// TIA Portal V16 export
// export: Created 2021-09-22T13:16:19.9691537Z, ExportSetting WithDefaults, DisplayName Totally Integrated Automation Portal, DisplayVersion V16 Update 1, DisplayName TIA Portal Version Control Interface, DisplayVersion V16, DisplayName TIA Portal Openness, DisplayVersion V16, DisplayName SINAMICS Startdrive Advanced, DisplayVersion V16 Update 5, DisplayName SINAMICS Startdrive G130, G150, S120, S150, SINAMICS MV, S210, DisplayVersion V16 Update 5, DisplayName SINAMICS Startdrive G110M, G120, G120C, G120D, G120P, G115D, DisplayVersion V16 Update 5, DisplayName STEP 7 Professional, DisplayVersion V16, DisplayName STEP 7 Safety, DisplayVersion V16, DisplayName WinCC Professional, DisplayVersion V16
FUNCTION_BLOCK "FB549.Divert.Sorter.Basing"   // FB543, LAD
{ S7_Optimized_Access := 'TRUE' }
VERSION : 0.1
// stored: AutoNumber false, IsIECCheckEnabled false, IsRetainMemResEnabled false, MemoryReserve 100, SetENOAutomatically false, UDAEnableTagReadback false
   VAR_INPUT
      Acil_Yok : Bool;
      Sorter_Calisiyor : Bool;
      Sağ_Chute_Sorted_Sensoru : Bool;
      Sol_Chute_Sorted_Sensoru : Bool;
      "Sağ_Chute_Aktif / Pasif" : Bool;   // 1 = Aktif , 0 = Pasif
      "Sol_Chute_Aktif / Pasif" : Bool;   // 1 = Aktif , 0 = Pasif
      Chute_Rulo_Hatası : Bool;
      Divert_Sürücü_Hatası : Bool;
      Pozisyon_Olcme_Aktif : Bool;
      Sağ_Çıkış_Target { ExternalAccessible := 'False'; ExternalVisible := 'False'; ExternalWritable := 'False'} : Int;
      Sol_Çıkış_Target { ExternalAccessible := 'False'; ExternalVisible := 'False'; ExternalWritable := 'False'} : Int;
      CN_NO : Int;
      "Aktüel Encoder Değeri" : LReal;
      Birinci_Divert_Min : LReal;
      Birinci_Divert_Max : LReal;
      İkinci_Divert_Min : LReal;
      İkinci_Divert_Max : LReal;
      Max_Kutu_Adedi { ExternalAccessible := 'False'; ExternalVisible := 'False'; ExternalWritable := 'False'} : Int;
   END_VAR
   VAR_OUTPUT
      "1_sol_Divert_Çalıştır" : Bool;
      "2_sol_Divert_Çalıştır" : Bool;
      "1_sağ_Divert_Çalıştır" : Bool;
      "2_sağ_Divert_Çalıştır" : Bool;
      "Sort Hatası" : Bool;
   END_VAR
   VAR
      Sort_Aktif_AUX : Array[1..10] of Bool;
      Sort_Aktif_PTrig : Array[1..10] of Bool;
      TOF_TIME : Array[1..10] of TOF_TIME;
      TON_TIME { S7_SetPoint := 'True'} : Array[1..10] of TON_TIME;
      Sort_Aktif1 : Bool;
      Sort_Aktif2 : Bool;
      Sort_Aktif1_Sağ : Bool;
      Sort_Aktif2_Sağ : Bool;
      Sağ_Sort_Pasif : Bool;
      Sol_Sort_Pasif : Bool;
      Ikinci_Servo_Baslama : Time;
      Divert_Durdur : Bool;
      Sort_Aktif_1 { ExternalAccessible := 'False'; ExternalVisible := 'False'; ExternalWritable := 'False'} : Array[1..10] of Bool;
      Sort_Aktif_2 { ExternalAccessible := 'False'; ExternalVisible := 'False'; ExternalWritable := 'False'} : Array[1..10] of Bool;
      Sort_Aktif_1_Sağ : Array[1..10] of Bool;
      Sort_Aktif_2_Sağ : Array[1..10] of Bool;
      Sort_Ilk_Pozisyon { ExternalAccessible := 'False'; ExternalVisible := 'False'; ExternalWritable := 'False'} : Array[1..10] of LReal;
      Sort_Ön_Pozisyon { ExternalAccessible := 'False'; ExternalVisible := 'False'; ExternalWritable := 'False'} : Array[1..10] of LReal;
      Sort_Aktif_Boy { ExternalAccessible := 'False'; ExternalVisible := 'False'; ExternalWritable := 'False'} : Array[1..10] of LReal;
      SortKutuNo : Int;
      Target100 : Bool;
      Target200 : Bool;
   END_VAR
   VAR_TEMP
      "On/Off" : Bool;
      j : Int;
      Ekstra_Uzunluk : LReal;
   END_VAR
   VAR_TEMP   // added for the SCL form of the ladder/FBD networks
      _w1 : Bool;
      _w2 : Bool;
      _w3 : Bool;
      _w4 : Bool;
   END_VAR
BEGIN

REGION Network 1: On / Off
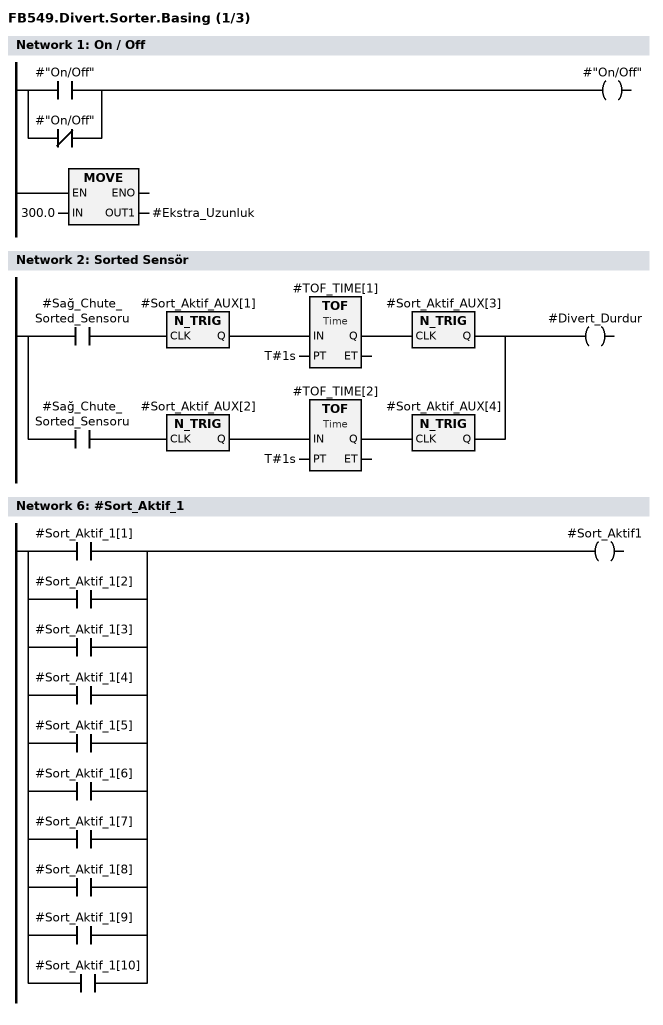
   RUNG wire#powerrail
      Contact( #"On/Off" )
      wire#w1
      Coil( #"On/Off" )
   END_RUNG
   RUNG wire#powerrail
      I_Contact( #"On/Off" )
   END_RUNG wire#w1
   RUNG wire#powerrail
      Move(in := 300.0, out1 => #Ekstra_Uzunluk)
   END_RUNG
   // the same network as SCL:
   #"On/Off" := #"On/Off" OR NOT #"On/Off";
   #Ekstra_Uzunluk := 300.0;
END_REGION

REGION Network 2: Sorted Sensör
   RUNG wire#powerrail
      Contact( #Sağ_Chute_Sorted_Sensoru )
      N_Trig( #Sort_Aktif_AUX[1] )
      { S7_Templates := "time_type := Time" } #TOF_TIME[1].TOF(pt := T#1s, et =>)
      N_Trig( #Sort_Aktif_AUX[3] )
      wire#w1
      Coil( #Divert_Durdur )
   END_RUNG
   RUNG wire#powerrail
      Contact( #Sağ_Chute_Sorted_Sensoru )
      N_Trig( #Sort_Aktif_AUX[2] )
      { S7_Templates := "time_type := Time" } #TOF_TIME[2].TOF(pt := T#1s, et =>)
      N_Trig( #Sort_Aktif_AUX[4] )
   END_RUNG wire#w1
   // the same network as SCL:
   #_w1 := NOT #Sağ_Chute_Sorted_Sensoru AND #Sort_Aktif_AUX[1];   // falling edge
   #Sort_Aktif_AUX[1] := #Sağ_Chute_Sorted_Sensoru;
   #TOF_TIME[1].TOF(IN := #_w1, PT := T#1s);
   #_w2 := NOT #TOF_TIME[1].Q AND #Sort_Aktif_AUX[3];   // falling edge
   #Sort_Aktif_AUX[3] := #TOF_TIME[1].Q;
   #_w3 := NOT #Sağ_Chute_Sorted_Sensoru AND #Sort_Aktif_AUX[2];   // falling edge
   #Sort_Aktif_AUX[2] := #Sağ_Chute_Sorted_Sensoru;
   #TOF_TIME[2].TOF(IN := #_w3, PT := T#1s);
   #_w4 := NOT #TOF_TIME[2].Q AND #Sort_Aktif_AUX[4];   // falling edge
   #Sort_Aktif_AUX[4] := #TOF_TIME[2].Q;
   #Divert_Durdur := #_w2 OR #_w4;
END_REGION

REGION Network 3 (SCL): Kutu Ön Arka Pozisyon Hesap
   // IF #Sensör.Sensor_N_Trig THEN
   //     #Sort_Ilk_Pozisyon["DB530_Kutu".CN_NO_Anlık_Kutu_Sayısı[#CN_NO]] := #"Aktüel Encoder Değeri";
   // END_IF;
   // FOR #j := 1 TO #Max_Kutu_Adedi BY 1 DO
   //     IF "DB530_Kutu".CN_NO[#CN_NO].Kutu_No[#j].VARMI = TRUE THEN
   //         #Sort_Ön_Pozisyon[#j] := #"Aktüel Encoder Değeri" - #Sort_Ilk_Pozisyon[#j];
   //     END_IF;
   // END_FOR;
END_REGION

REGION Network 4 (SCL): Sol Sort Aktif Kararı
   IF #Pozisyon_Olcme_Aktif = 0
       // AND #Sorter_Calisiyor = TRUE
       // AND #"Sol_Chute_Aktif / Pasif"
   THEN
       FOR #j := 1 TO #Max_Kutu_Adedi BY 1 DO
           IF "DB530_Kutu".CN_NO[#CN_NO].Kutu_No[#j].VARMI THEN

               IF "DB530_Kutu".CN_NO[#CN_NO].Kutu_No[#j].Target = 201
                   OR "DB530_Kutu".CN_NO[#CN_NO].Kutu_No[#j].Target = 202
                   OR "DB530_Kutu".CN_NO[#CN_NO].Kutu_No[#j].Target = 203
                   OR "DB530_Kutu".CN_NO[#CN_NO].Kutu_No[#j].Target = 204 THEN
                   #Target200 := 1;
               ELSE
                   #Target200 := 0;
               END_IF;

               IF #"Sol_Chute_Aktif / Pasif" = 1
                   AND #Chute_Rulo_Hatası = 0
                   AND #Divert_Sürücü_Hatası = 0
                   // AND #Sol_Sort_Pasif = 0
                   AND #Acil_Yok = 1
                   AND "DB530_Kutu".CN_NO[#CN_NO].Kutu_No[#j].Posizyon >= #Birinci_Divert_Min
                   AND "DB530_Kutu".CN_NO[#CN_NO].Kutu_No[#j].Posizyon <= #Birinci_Divert_Min + "DB530_Kutu".CN_NO[#CN_NO].Kutu_No[#j].Uzunluk + #Ekstra_Uzunluk
                   AND  #Target200 = 1
                   // AND "DB530_Kutu".CN_NO[#CN_NO].Kutu_No[#j].Sort_Aktifleştirildi = FALSE
               THEN
                   #Sort_Aktif_1[#j] := TRUE;
               ELSE
                   #Sort_Aktif_1[#j] := FALSE;
               END_IF;

               IF #"Sol_Chute_Aktif / Pasif" = 1
                   AND #Chute_Rulo_Hatası = 0
                   AND #Divert_Sürücü_Hatası = 0
                   // AND #Sol_Sort_Pasif = 0
                   AND #Acil_Yok = 1
                   AND "DB530_Kutu".CN_NO[#CN_NO].Kutu_No[#j].Posizyon >= #İkinci_Divert_Min
                   AND "DB530_Kutu".CN_NO[#CN_NO].Kutu_No[#j].Posizyon <= #İkinci_Divert_Min + "DB530_Kutu".CN_NO[#CN_NO].Kutu_No[#j].Uzunluk + #Ekstra_Uzunluk
                   AND #Target200 = 1
                   // AND "DB530_Kutu".CN_NO[#CN_NO].Kutu_No[#j].Sort_Aktifleştirildi = FALSE
               THEN
                   #Sort_Aktif_2[#j] := TRUE;
               ELSE
                   #Sort_Aktif_2[#j] := FALSE;
               END_IF;

               // IF "DB530_Kutu".CN_NO[#CN_NO].Kutu_No[#j].Posizyon > #İkinci_Divert_Max + "DB530_Kutu".CN_NO[#CN_NO].Kutu_No[#j].Uzunluk THEN
               //     "DB530_Kutu".CN_NO[#CN_NO].Kutu_No[#j].Sort_Aktifleştirildi := true;
               // END_IF;

               ///////////SortStatus//SolTaraf
               IF #Target200 = 1 // Sol Çıkış Statüleri
                   // AND "DB530_Kutu".CN_NO[#CN_NO].Kutu_No[#j].VARMI = True
                   AND ("DB530_Kutu".CN_NO[#CN_NO].Kutu_No[#j].Posizyon >= #Birinci_Divert_Min OR "DB530_Kutu".CN_NO[#CN_NO].Kutu_No[#j].Posizyon >= #İkinci_Divert_Min)
                   // AND "DB530_Kutu".CN_NO[#CN_NO].Kutu_No[#j].Sort_Aktifleştirildi = 0
                   // AND (#"Sol_Chute_Aktif / Pasif" = 0 OR #Divert_Sürücü_Hatası = 1 OR #Chute_Rulo_Hatası = 1)
               THEN
                   IF #"Sol_Chute_Aktif / Pasif" = 0 OR #Acil_Yok = 0 THEN
                       "DB530_Kutu".CN_NO[#CN_NO].Kutu_No[#j].Sort_Statu := 1;
                       // "DB530_Kutu".CN_NO[#CN_NO].Kutu_No[#j].Sort_Aktifleştirildi := 1;
                   ELSIF #Divert_Sürücü_Hatası = 1 THEN
                       "DB530_Kutu".CN_NO[#CN_NO].Kutu_No[#j].Sort_Statu := 2;
                       // "DB530_Kutu".CN_NO[#CN_NO].Kutu_No[#j].Sort_Aktifleştirildi := 1;
                   ELSIF #Chute_Rulo_Hatası = 1 THEN
                       "DB530_Kutu".CN_NO[#CN_NO].Kutu_No[#j].Sort_Statu := 3;
                       // "DB530_Kutu".CN_NO[#CN_NO].Kutu_No[#j].Sort_Aktifleştirildi := 1;
                   ELSIF (#Sort_Aktif_1[#j] = 1 OR #Sort_Aktif_2[#j] = 1) THEN
                       "DB530_Kutu".CN_NO[#CN_NO].Kutu_No[#j].Sort_Statu := 10;
                       "DB530_Kutu".CN_NO[#CN_NO].Kutu_No[#j].Sort_Aktifleştirildi := 1;
                       "DB542.Chute.Kontrol".CN_NO[#CN_NO].Sort_UID_Kutu_No[#j] := "DB530_Kutu".CN_NO[#CN_NO].Kutu_No[#j].UniqueID;
                   END_IF;
               END_IF;
           END_IF;
           IF "DB530_Kutu".CN_NO[#CN_NO].Kutu_No[1].VARMI = 0 THEN
               #Sort_Aktif_1[#j] := FALSE;
               #Sort_Aktif_2[#j] := FALSE;
           END_IF;
       END_FOR;
   END_IF;
END_REGION

REGION Network 5 (SCL): Sağ Sort Aktif Kararı
   IF #Pozisyon_Olcme_Aktif = 0
       // AND #Sorter_Calisiyor = TRUE
       // AND #"Sağ_Chute_Aktif / Pasif"
   THEN

       FOR #j := 1 TO #Max_Kutu_Adedi BY 1 DO
           IF "DB530_Kutu".CN_NO[#CN_NO].Kutu_No[#j].VARMI THEN

               IF     "DB530_Kutu".CN_NO[#CN_NO].Kutu_No[#j].Target = 101
                   OR "DB530_Kutu".CN_NO[#CN_NO].Kutu_No[#j].Target = 102
                   OR "DB530_Kutu".CN_NO[#CN_NO].Kutu_No[#j].Target = 103
                   OR "DB530_Kutu".CN_NO[#CN_NO].Kutu_No[#j].Target = 104 THEN
                   #Target100 := 1;
               ELSE
                   #Target100 := 0;
               END_IF;

               IF #"Sağ_Chute_Aktif / Pasif" = 1
                   AND #Chute_Rulo_Hatası = 0
                   AND #Divert_Sürücü_Hatası = 0
                   // AND #Sağ_Sort_Pasif = 0
                   AND #Acil_Yok = 1
                   AND "DB530_Kutu".CN_NO[#CN_NO].Kutu_No[#j].Posizyon >= #Birinci_Divert_Min
                   AND "DB530_Kutu".CN_NO[#CN_NO].Kutu_No[#j].Posizyon <= #Birinci_Divert_Min + "DB530_Kutu".CN_NO[#CN_NO].Kutu_No[#j].Uzunluk + #Ekstra_Uzunluk
                   AND #Target100 = 1
                   // AND "DB530_Kutu".CN_NO[#CN_NO].Kutu_No[#j].Sort_Aktifleştirildi = FALSE
               THEN
                   #Sort_Aktif_1_Sağ[#j] := TRUE;
               ELSE
                   #Sort_Aktif_1_Sağ[#j] := FALSE;
               END_IF;

               IF #"Sağ_Chute_Aktif / Pasif" = 1
                   AND #Chute_Rulo_Hatası = 0
                   AND #Divert_Sürücü_Hatası = 0
                   // AND #Sağ_Sort_Pasif = 0
                   AND #Acil_Yok = 1
                   AND "DB530_Kutu".CN_NO[#CN_NO].Kutu_No[#j].Posizyon >= #İkinci_Divert_Min
                   AND "DB530_Kutu".CN_NO[#CN_NO].Kutu_No[#j].Posizyon <= #İkinci_Divert_Min + "DB530_Kutu".CN_NO[#CN_NO].Kutu_No[#j].Uzunluk + #Ekstra_Uzunluk
                   AND #Target100 = 1
                   // AND "DB530_Kutu".CN_NO[#CN_NO].Kutu_No[#j].Sort_Aktifleştirildi = FALSE
               THEN
                   #Sort_Aktif_2_Sağ[#j] := TRUE;
               ELSE
                   #Sort_Aktif_2_Sağ[#j] := FALSE;
               END_IF;

               // IF "DB530_Kutu".CN_NO[#CN_NO].Kutu_No[#j].Posizyon > #İkinci_Divert_Max + "DB530_Kutu".CN_NO[#CN_NO].Kutu_No[#j].Uzunluk THEN
               //     "DB530_Kutu".CN_NO[#CN_NO].Kutu_No[#j].Sort_Aktifleştirildi := true;
               // END_IF;

               ///////////SortStatus//SağTaraf
               IF #Target100 = 1 // Sağ Çıkış Statüleri
                   // AND "DB530_Kutu".CN_NO[#CN_NO].Kutu_No[#j].VARMI = True
                   AND ("DB530_Kutu".CN_NO[#CN_NO].Kutu_No[#j].Posizyon >= #Birinci_Divert_Min OR "DB530_Kutu".CN_NO[#CN_NO].Kutu_No[#j].Posizyon >= #İkinci_Divert_Min)
                   // AND "DB530_Kutu".CN_NO[#CN_NO].Kutu_No[#j].Sort_Aktifleştirildi = 0
                   // AND (#"Sağ_Chute_Aktif / Pasif" = 0 OR #Divert_Sürücü_Hatası = 1 OR #Chute_Rulo_Hatası = 1)
               THEN
                   IF #"Sağ_Chute_Aktif / Pasif" = 0 OR #Acil_Yok = 0 THEN
                       "DB530_Kutu".CN_NO[#CN_NO].Kutu_No[#j].Sort_Statu := 1;
                       // "DB530_Kutu".CN_NO[#CN_NO].Kutu_No[#j].Sort_Aktifleştirildi := 1;
                   ELSIF #Divert_Sürücü_Hatası = 1 THEN
                       "DB530_Kutu".CN_NO[#CN_NO].Kutu_No[#j].Sort_Statu := 2;
                       // "DB530_Kutu".CN_NO[#CN_NO].Kutu_No[#j].Sort_Aktifleştirildi := 1;
                   ELSIF #Chute_Rulo_Hatası = 1 THEN
                       "DB530_Kutu".CN_NO[#CN_NO].Kutu_No[#j].Sort_Statu := 3;
                       // "DB530_Kutu".CN_NO[#CN_NO].Kutu_No[#j].Sort_Aktifleştirildi := 1;
                   ELSIF (#Sort_Aktif_1_Sağ[#j] = 1 OR #Sort_Aktif_2_Sağ[#j] = 1) THEN
                       "DB530_Kutu".CN_NO[#CN_NO].Kutu_No[#j].Sort_Statu := 10;
                       "DB530_Kutu".CN_NO[#CN_NO].Kutu_No[#j].Sort_Aktifleştirildi := 1;
                       "DB542.Chute.Kontrol".CN_NO[#CN_NO].Sort_UID_Kutu_No[#j] := "DB530_Kutu".CN_NO[#CN_NO].Kutu_No[#j].UniqueID;
                   END_IF;
               END_IF;
           END_IF;
           IF "DB530_Kutu".CN_NO[#CN_NO].Kutu_No[1].VARMI = 0 THEN
               #Sort_Aktif_1_Sağ[#j] := FALSE;
               #Sort_Aktif_2_Sağ[#j] := FALSE;
           END_IF;
       END_FOR;
   END_IF;
END_REGION

REGION Network 6: #Sort_Aktif_1
   RUNG wire#powerrail
      Contact( #Sort_Aktif_1[1] )
      wire#w1
      Coil( #Sort_Aktif1 )
   END_RUNG
   RUNG wire#powerrail
      Contact( #Sort_Aktif_1[2] )
   END_RUNG wire#w1
   RUNG wire#powerrail
      Contact( #Sort_Aktif_1[3] )
   END_RUNG wire#w1
   RUNG wire#powerrail
      Contact( #Sort_Aktif_1[4] )
   END_RUNG wire#w1
   RUNG wire#powerrail
      Contact( #Sort_Aktif_1[5] )
   END_RUNG wire#w1
   RUNG wire#powerrail
      Contact( #Sort_Aktif_1[6] )
   END_RUNG wire#w1
   RUNG wire#powerrail
      Contact( #Sort_Aktif_1[7] )
   END_RUNG wire#w1
   RUNG wire#powerrail
      Contact( #Sort_Aktif_1[8] )
   END_RUNG wire#w1
   RUNG wire#powerrail
      Contact( #Sort_Aktif_1[9] )
   END_RUNG wire#w1
   RUNG wire#powerrail
      Contact( #Sort_Aktif_1[10] )
   END_RUNG wire#w1
   // the same network as SCL:
   #Sort_Aktif1 := #Sort_Aktif_1[1] OR #Sort_Aktif_1[2] OR #Sort_Aktif_1[3] OR #Sort_Aktif_1[4] OR #Sort_Aktif_1[5] OR #Sort_Aktif_1[6] OR #Sort_Aktif_1[7] OR #Sort_Aktif_1[8] OR #Sort_Aktif_1[9] OR #Sort_Aktif_1[10];
END_REGION

REGION Network 7: #Sort_Aktif_2
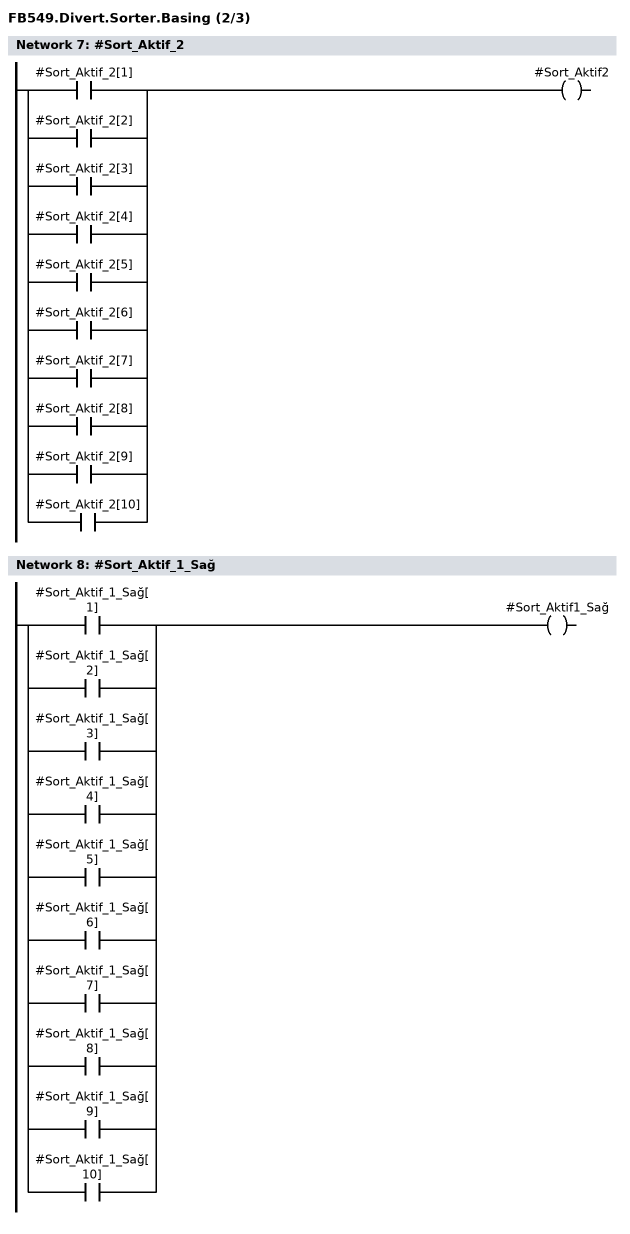
   RUNG wire#powerrail
      Contact( #Sort_Aktif_2[1] )
      wire#w1
      Coil( #Sort_Aktif2 )
   END_RUNG
   RUNG wire#powerrail
      Contact( #Sort_Aktif_2[2] )
   END_RUNG wire#w1
   RUNG wire#powerrail
      Contact( #Sort_Aktif_2[3] )
   END_RUNG wire#w1
   RUNG wire#powerrail
      Contact( #Sort_Aktif_2[4] )
   END_RUNG wire#w1
   RUNG wire#powerrail
      Contact( #Sort_Aktif_2[5] )
   END_RUNG wire#w1
   RUNG wire#powerrail
      Contact( #Sort_Aktif_2[6] )
   END_RUNG wire#w1
   RUNG wire#powerrail
      Contact( #Sort_Aktif_2[7] )
   END_RUNG wire#w1
   RUNG wire#powerrail
      Contact( #Sort_Aktif_2[8] )
   END_RUNG wire#w1
   RUNG wire#powerrail
      Contact( #Sort_Aktif_2[9] )
   END_RUNG wire#w1
   RUNG wire#powerrail
      Contact( #Sort_Aktif_2[10] )
   END_RUNG wire#w1
   // the same network as SCL:
   #Sort_Aktif2 := #Sort_Aktif_2[1] OR #Sort_Aktif_2[2] OR #Sort_Aktif_2[3] OR #Sort_Aktif_2[4] OR #Sort_Aktif_2[5] OR #Sort_Aktif_2[6] OR #Sort_Aktif_2[7] OR #Sort_Aktif_2[8] OR #Sort_Aktif_2[9] OR #Sort_Aktif_2[10];
END_REGION

REGION Network 8: #Sort_Aktif_1_Sağ
   RUNG wire#powerrail
      Contact( #Sort_Aktif_1_Sağ[1] )
      wire#w1
      Coil( #Sort_Aktif1_Sağ )
   END_RUNG
   RUNG wire#powerrail
      Contact( #Sort_Aktif_1_Sağ[2] )
   END_RUNG wire#w1
   RUNG wire#powerrail
      Contact( #Sort_Aktif_1_Sağ[3] )
   END_RUNG wire#w1
   RUNG wire#powerrail
      Contact( #Sort_Aktif_1_Sağ[4] )
   END_RUNG wire#w1
   RUNG wire#powerrail
      Contact( #Sort_Aktif_1_Sağ[5] )
   END_RUNG wire#w1
   RUNG wire#powerrail
      Contact( #Sort_Aktif_1_Sağ[6] )
   END_RUNG wire#w1
   RUNG wire#powerrail
      Contact( #Sort_Aktif_1_Sağ[7] )
   END_RUNG wire#w1
   RUNG wire#powerrail
      Contact( #Sort_Aktif_1_Sağ[8] )
   END_RUNG wire#w1
   RUNG wire#powerrail
      Contact( #Sort_Aktif_1_Sağ[9] )
   END_RUNG wire#w1
   RUNG wire#powerrail
      Contact( #Sort_Aktif_1_Sağ[10] )
   END_RUNG wire#w1
   // the same network as SCL:
   #Sort_Aktif1_Sağ := #Sort_Aktif_1_Sağ[1] OR #Sort_Aktif_1_Sağ[2] OR #Sort_Aktif_1_Sağ[3] OR #Sort_Aktif_1_Sağ[4] OR #Sort_Aktif_1_Sağ[5] OR #Sort_Aktif_1_Sağ[6] OR #Sort_Aktif_1_Sağ[7] OR #Sort_Aktif_1_Sağ[8] OR #Sort_Aktif_1_Sağ[9] OR #Sort_Aktif_1_Sağ[10];
END_REGION

REGION Network 9: #Sort_Aktif_2_Sağ
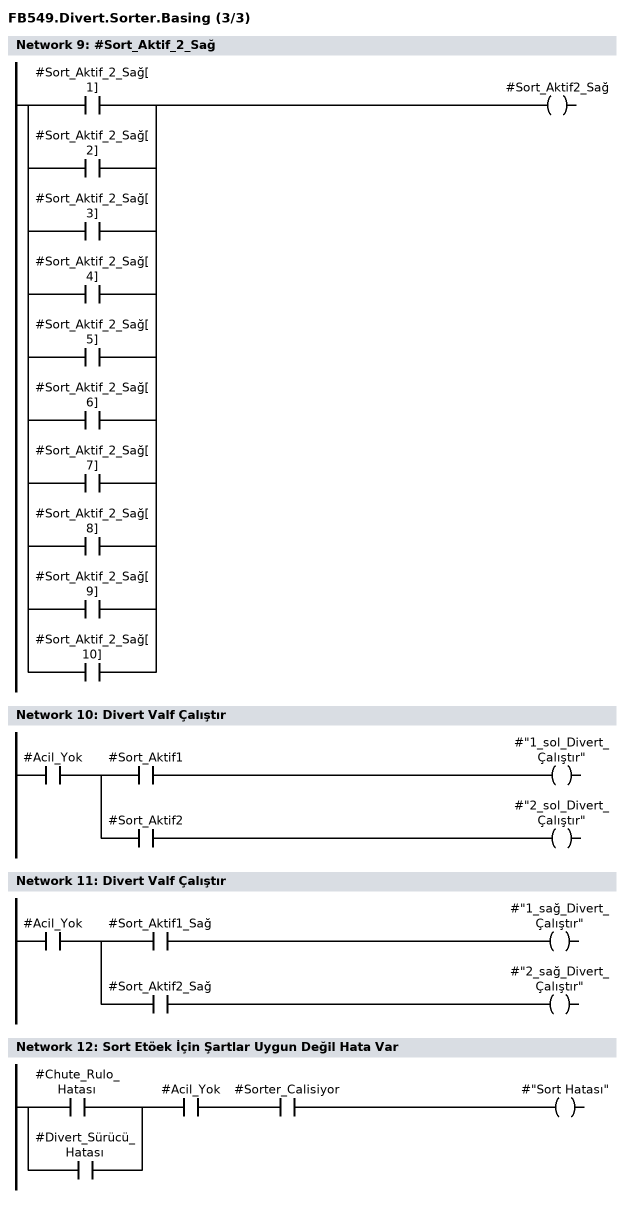
   RUNG wire#powerrail
      Contact( #Sort_Aktif_2_Sağ[1] )
      wire#w1
      Coil( #Sort_Aktif2_Sağ )
   END_RUNG
   RUNG wire#powerrail
      Contact( #Sort_Aktif_2_Sağ[2] )
   END_RUNG wire#w1
   RUNG wire#powerrail
      Contact( #Sort_Aktif_2_Sağ[3] )
   END_RUNG wire#w1
   RUNG wire#powerrail
      Contact( #Sort_Aktif_2_Sağ[4] )
   END_RUNG wire#w1
   RUNG wire#powerrail
      Contact( #Sort_Aktif_2_Sağ[5] )
   END_RUNG wire#w1
   RUNG wire#powerrail
      Contact( #Sort_Aktif_2_Sağ[6] )
   END_RUNG wire#w1
   RUNG wire#powerrail
      Contact( #Sort_Aktif_2_Sağ[7] )
   END_RUNG wire#w1
   RUNG wire#powerrail
      Contact( #Sort_Aktif_2_Sağ[8] )
   END_RUNG wire#w1
   RUNG wire#powerrail
      Contact( #Sort_Aktif_2_Sağ[9] )
   END_RUNG wire#w1
   RUNG wire#powerrail
      Contact( #Sort_Aktif_2_Sağ[10] )
   END_RUNG wire#w1
   // the same network as SCL:
   #Sort_Aktif2_Sağ := #Sort_Aktif_2_Sağ[1] OR #Sort_Aktif_2_Sağ[2] OR #Sort_Aktif_2_Sağ[3] OR #Sort_Aktif_2_Sağ[4] OR #Sort_Aktif_2_Sağ[5] OR #Sort_Aktif_2_Sağ[6] OR #Sort_Aktif_2_Sağ[7] OR #Sort_Aktif_2_Sağ[8] OR #Sort_Aktif_2_Sağ[9] OR #Sort_Aktif_2_Sağ[10];
END_REGION

REGION Network 10: Divert Valf Çalıştır
   RUNG wire#powerrail
      Contact( #Acil_Yok )
      wire#w1
      Contact( #Sort_Aktif1 )
      Coil( #"1_sol_Divert_Çalıştır" )
   END_RUNG
   RUNG wire#w1
      Contact( #Sort_Aktif2 )
      Coil( #"2_sol_Divert_Çalıştır" )
   END_RUNG
   // the same network as SCL:
   #"1_sol_Divert_Çalıştır" := #Acil_Yok AND #Sort_Aktif1;
   #"2_sol_Divert_Çalıştır" := #Acil_Yok AND #Sort_Aktif2;
END_REGION

REGION Network 11: Divert Valf Çalıştır
   RUNG wire#powerrail
      Contact( #Acil_Yok )
      wire#w1
      Contact( #Sort_Aktif1_Sağ )
      Coil( #"1_sağ_Divert_Çalıştır" )
   END_RUNG
   RUNG wire#w1
      Contact( #Sort_Aktif2_Sağ )
      Coil( #"2_sağ_Divert_Çalıştır" )
   END_RUNG
   // the same network as SCL:
   #"1_sağ_Divert_Çalıştır" := #Acil_Yok AND #Sort_Aktif1_Sağ;
   #"2_sağ_Divert_Çalıştır" := #Acil_Yok AND #Sort_Aktif2_Sağ;
END_REGION

REGION Network 12: Sort Etöek İçin Şartlar Uygun Değil Hata Var
   RUNG wire#powerrail
      Contact( #Chute_Rulo_Hatası )
      wire#w1
      Contact( #Acil_Yok )
      Contact( #Sorter_Calisiyor )
      Coil( #"Sort Hatası" )
   END_RUNG
   RUNG wire#powerrail
      Contact( #Divert_Sürücü_Hatası )
   END_RUNG wire#w1
   // the same network as SCL:
   #"Sort Hatası" := (#Chute_Rulo_Hatası OR #Divert_Sürücü_Hatası) AND #Acil_Yok AND #Sorter_Calisiyor;
END_REGION
END_FUNCTION_BLOCK
